// Mitsubishi GX Works2 project: practice2   PLC: Q03UDV

PROGRAM MAIN
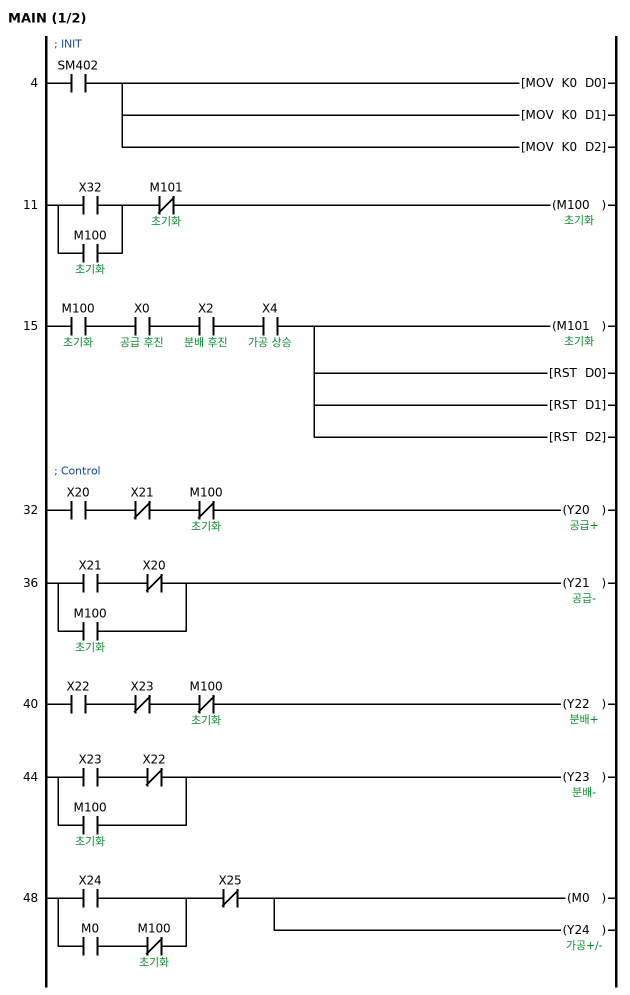
; INIT
4     LD      SM402
      MOV     K0 D0
      MOV     K0 D1
      MOV     K0 D2
11    LD      X32
      OR      M100  ; 초기화
      ANI     M101  ; 초기화
      OUT     M100  ; 초기화
15    LD      M100  ; 초기화
      AND     X0  ; 공급 후진
      AND     X2  ; 분배 후진
      AND     X4  ; 가공 상승
      OUT     M101  ; 초기화
      RST     D0
      RST     D1
      RST     D2
; Control
32    LD      X20
      ANI     X21
      ANI     M100  ; 초기화
      OUT     Y20  ; 공급+
36    LD      X21
      ANI     X20
      OR      M100  ; 초기화
      OUT     Y21  ; 공급-
40    LD      X22
      ANI     X23
      ANI     M100  ; 초기화
      OUT     Y22  ; 분배+
44    LD      X23
      ANI     X22
      OR      M100  ; 초기화
      OUT     Y23  ; 분배-
48    LD      X24
      LD      M0
      ANI     M100  ; 초기화
      ORB
      ANI     X25
      OUT     M0
      OUT     Y24  ; 가공+/-
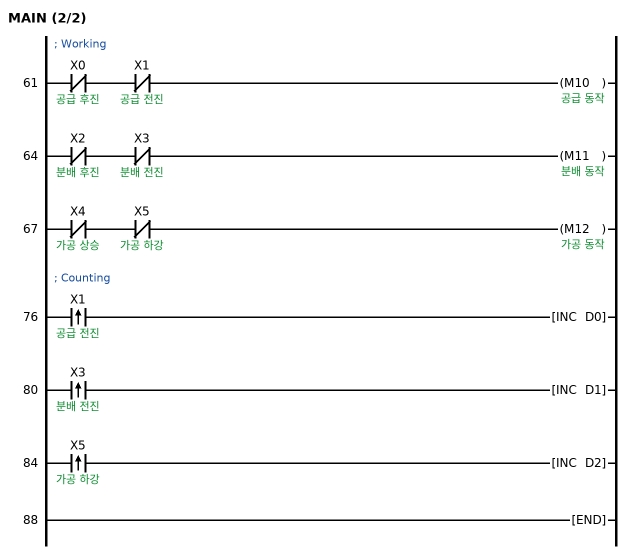
; Working
61    LDI     X0  ; 공급 후진
      ANI     X1  ; 공급 전진
      OUT     M10  ; 공급 동작
64    LDI     X2  ; 분배 후진
      ANI     X3  ; 분배 전진
      OUT     M11  ; 분배 동작
67    LDI     X4  ; 가공 상승
      ANI     X5  ; 가공 하강
      OUT     M12  ; 가공 동작
; Counting
76    LDP     X1  ; 공급 전진
      INC     D0
80    LDP     X3  ; 분배 전진
      INC     D1
84    LDP     X5  ; 가공 하강
      INC     D2
88    END
END_PROGRAM

// device comments not shown above
M200  ; 코멘트
